// TIA Portal V20 export
TYPE "zp_CITIData"
// stored: Access Published, Namespace CITI_Logic
   STRUCT
      EoC { S7_SetPoint := 'True'} : "CITI_Logic.zp_CITIEoC";
      CoS : "CITI_Logic.zp_CITICoS";
      TradeCall { S7_SetPoint := 'True'} : "CITI_Logic.zp_CITITradeCalls";
      FaultString { S7_SetPoint := 'True'} : String[200];
      Machine_Loading : Bool;
      Machine_Unloading : Bool;
      Machine_Processing : Bool;
      Shift_Reset : Bool;
      Clock_Sync : Bool;
      Dry_Cycle_Mode : Bool;
      CITI_DryCycle_Blocker : Bool;
      Control_Power_On : Bool;
      IT_Heartbeat : Bool;
      Write_Day : SInt;
      Write_Month : SInt;
      Write_Year : SInt;
      ShiftNumber : SInt;
      Current_Cycle_Time : DInt;
   END_STRUCT;
END_TYPE
